(* Logix 5000 project; controller LeakTestAuto vendor 1 type 14 code 226 rev 37.11; software revision 37.01; part 6 of 12 *)
(* tags used below, declared in another part *)
   AOI_CTS1 : AOI_CTS_INSTRUMENT;
   AOI_CTS2 : AOI_CTS_INSTRUMENT;
   AOI_OP220_Seq : AOI_Sequencer_x64;
   AOI_RobotPos : AOI_RobotPositions;
   AOI_SeqSteps : AOI_StandardSeqSteps;
   AOI_SRX100 : AOI_KeyenceBarcode;
   Barcode_ResultData : STR_Barcode;
   BarcodeBypass : BOOL;
   BarcodeInputs : udt_KeyenceScannerInputs;
   BarcodeScanner : udt_OutputStructure;
   Conveyor : udt_OutputStructure;
   Conveyor_Seq : udt_SequenceStructure_X64;
   ConveyorHomeCounter : COUNTER;
   CurrentDUTData : udt_DUTHistory[2];
   DryCycle_N1Ready : BOOL;
   DryCycle_N2Ready : BOOL;
   DUTHistoryDump : udt_DUTHistory;
   DUTTestHistory : udt_DUTHistory[10];
   FFLU_DUTHistory : CONTROL;
   InfeedCounter : COUNTER;
   LeakTester1 : udt_OutputStructure;
   LeakTester2 : udt_OutputStructure;
   Nest1Bypass : BOOL;
   Nest1Cylinder : udt_OutputStructure;
   Nest1Empty : BOOL;
   Nest1Ready : BOOL;
   Nest2Bypass : BOOL;
   Nest2Cylinder : udt_OutputStructure;
   Nest2Empty : BOOL;
   Nest2Ready : BOOL;
   OP220 : udt_Mode;
   OP220_HomingSeq : udt_SequenceStructure_X64;
   OP220_Seq : udt_SequenceStructure_X64;
   OutfeedCounter : COUNTER;
   ResetFeedCounters : BOOL;
   RFID_TagStatus : BOOL[32];
   RFIDLoadingNestScanner : udt_OutputStructure;
   RFIDScanner : udt_OutputStructure;
   Robot : udt_OutputStructure;
   RobotGripper : udt_OutputStructure;
   RobotInputs : udt_EpsonInputs;
   TON_ConvUnloadDelay : TIMER;
   Delay_TMR : TIMER[11];   // Delay Timers
   I_OP220_N3_CONVEYOR_LOAD : ALIAS FOR Local:3:I.Pt12.Data;
   I_OP220_N3_CONVEYOR_UNLOAD : ALIAS FOR Local:3:I.Pt14.Data;
   I_OP220_N3_DUT_PRE_NEST_0 : ALIAS FOR Local:3:I.Pt00.Data;
   I_OP220_N3_DUT_PRE_NEST_1 : ALIAS FOR Local:3:I.Pt01.Data;
   I_OP220_N3_DUT_PRE_NEST_2 : ALIAS FOR Local:3:I.Pt02.Data;
   I_OP220_N3_NEST1_EXTEND : ALIAS FOR Local:3:I.Pt04.Data;
   I_OP220_N3_NEST1_HOME : ALIAS FOR Local:3:I.Pt03.Data;
   I_OP220_N3_NEST2_EXTEND : ALIAS FOR Local:3:I.Pt06.Data;
   I_OP220_N3_NEST2_HOME : ALIAS FOR Local:3:I.Pt05.Data;
   Ignition_Bypass : BOOL;
   James_Dint : DINT;   // James Test Word
   null : STRING;
   PLC : AOI_PLC;
   ST1_Ignition_DataReady : BOOL;
   ST1_Ignition_DataReady_Setup : BOOL;
   ST1_Ignition_DataReceived : BOOL;
   ST1_Ignition_SerialNum : STRING;
   ST1_Ignition_Status : DINT;
   ST2_Ignition_DataReady : BOOL;
   ST2_Ignition_DataReady_Setup : BOOL;
   ST2_Ignition_DataReceived : BOOL;
   ST2_Ignition_SerialNum : STRING;
   ST2_Ignition_Status : DINT;
(* MainProgram, continued *)

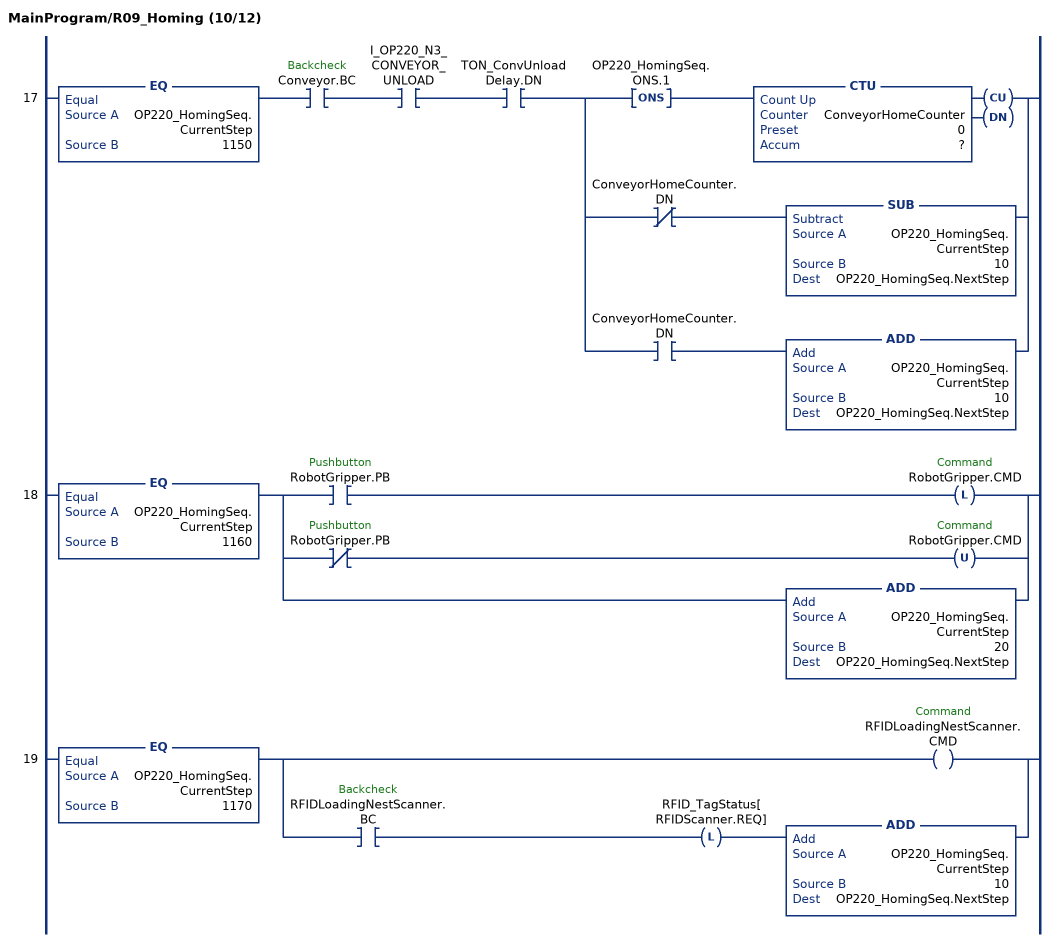
   [picture p62: MainProgram/R09_Homing rungs 17-19]
   17: EQ(OP220_HomingSeq.CurrentStep,1150)XIC(Conveyor.BC)XIC(I_OP220_N3_CONVEYOR_UNLOAD)XIC(TON_ConvUnloadDelay.DN)[ONS(OP220_HomingSeq.ONS.1) CTU(ConveyorHomeCounter,?,?) ,[XIO(ConveyorHomeCounter.DN) SUB(OP220_HomingSeq.CurrentStep,10,OP220_HomingSeq.NextStep) ,XIC(ConveyorHomeCounter.DN) ADD(OP220_HomingSeq.CurrentStep,10,OP220_HomingSeq.NextStep) ] ];
   18: EQ(OP220_HomingSeq.CurrentStep,1160)[XIC(RobotGripper.PB) OTL(RobotGripper.CMD) ,XIO(RobotGripper.PB) OTU(RobotGripper.CMD) ,ADD(OP220_HomingSeq.CurrentStep,20,OP220_HomingSeq.NextStep) ];
   19: EQ(OP220_HomingSeq.CurrentStep,1170)[OTE(RFIDLoadingNestScanner.CMD) ,XIC(RFIDLoadingNestScanner.BC) OTL(RFID_TagStatus[RFIDScanner.REQ]) ADD(OP220_HomingSeq.CurrentStep,10,OP220_HomingSeq.NextStep) ];
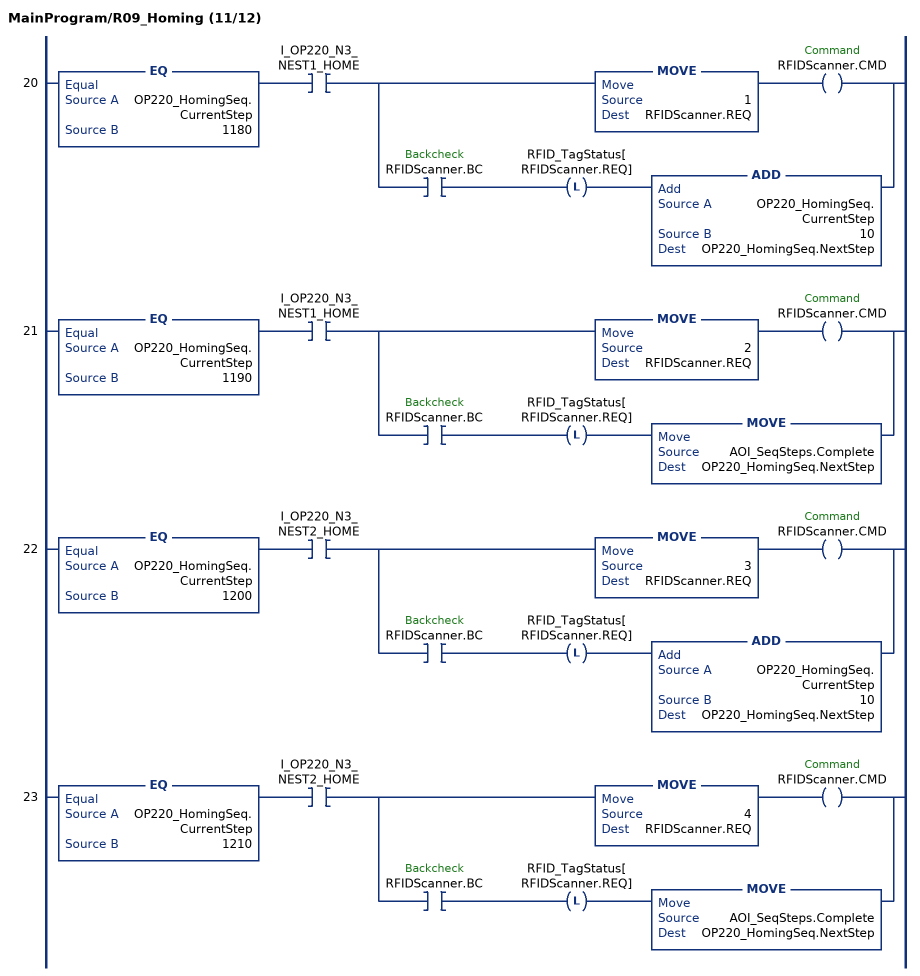
   20: EQ(OP220_HomingSeq.CurrentStep,1180)XIC(I_OP220_N3_NEST1_HOME)[MOVE(1,RFIDScanner.REQ) OTE(RFIDScanner.CMD) ,XIC(RFIDScanner.BC) OTL(RFID_TagStatus[RFIDScanner.REQ]) ADD(OP220_HomingSeq.CurrentStep,10,OP220_HomingSeq.NextStep) ];
   21: EQ(OP220_HomingSeq.CurrentStep,1190)XIC(I_OP220_N3_NEST1_HOME)[MOVE(2,RFIDScanner.REQ) OTE(RFIDScanner.CMD) ,XIC(RFIDScanner.BC) OTL(RFID_TagStatus[RFIDScanner.REQ]) MOVE(AOI_SeqSteps.Complete,OP220_HomingSeq.NextStep) ];
   22: EQ(OP220_HomingSeq.CurrentStep,1200)XIC(I_OP220_N3_NEST2_HOME)[MOVE(3,RFIDScanner.REQ) OTE(RFIDScanner.CMD) ,XIC(RFIDScanner.BC) OTL(RFID_TagStatus[RFIDScanner.REQ]) ADD(OP220_HomingSeq.CurrentStep,10,OP220_HomingSeq.NextStep) ];
   23: EQ(OP220_HomingSeq.CurrentStep,1210)XIC(I_OP220_N3_NEST2_HOME)[MOVE(4,RFIDScanner.REQ) OTE(RFIDScanner.CMD) ,XIC(RFIDScanner.BC) OTL(RFID_TagStatus[RFIDScanner.REQ]) MOVE(AOI_SeqSteps.Complete,OP220_HomingSeq.NextStep) ];
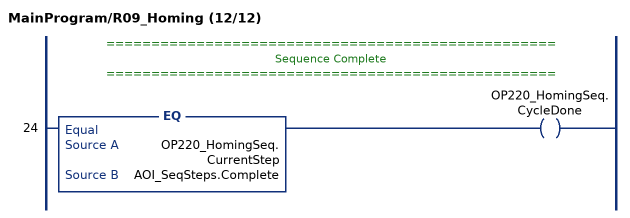
   // ==================================================
   // Sequence Complete
   // ==================================================
   24: EQ(OP220_HomingSeq.CurrentStep,AOI_SeqSteps.Complete)OTE(OP220_HomingSeq.CycleDone);
END_ROUTINE

ROUTINE R10_Sequence   (* ladder *)
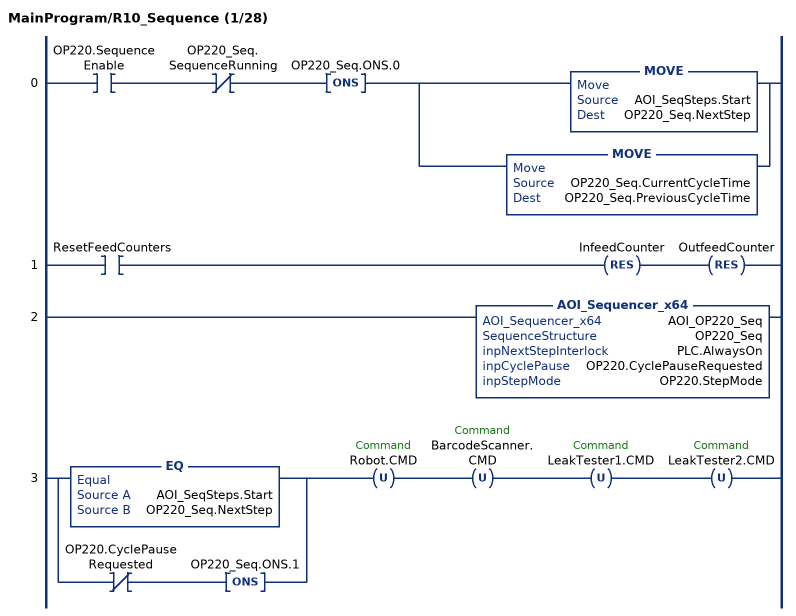
   0: XIC(OP220.SequenceEnable)XIO(OP220_Seq.SequenceRunning)ONS(OP220_Seq.ONS.0)[MOVE(AOI_SeqSteps.Start,OP220_Seq.NextStep) ,MOVE(OP220_Seq.CurrentCycleTime,OP220_Seq.PreviousCycleTime) ];
   1: XIC(ResetFeedCounters)RES(InfeedCounter)RES(OutfeedCounter);
   2: AOI_Sequencer_x64(AOI_OP220_Seq,OP220_Seq,PLC.AlwaysOn,OP220.CyclePauseRequested,OP220.StepMode);
   3: [EQ(AOI_SeqSteps.Start,OP220_Seq.NextStep) ,XIO(OP220.CyclePauseRequested) ONS(OP220_Seq.ONS.1) ]OTU(Robot.CMD)OTU(BarcodeScanner.CMD)OTU(LeakTester1.CMD)OTU(LeakTester2.CMD);
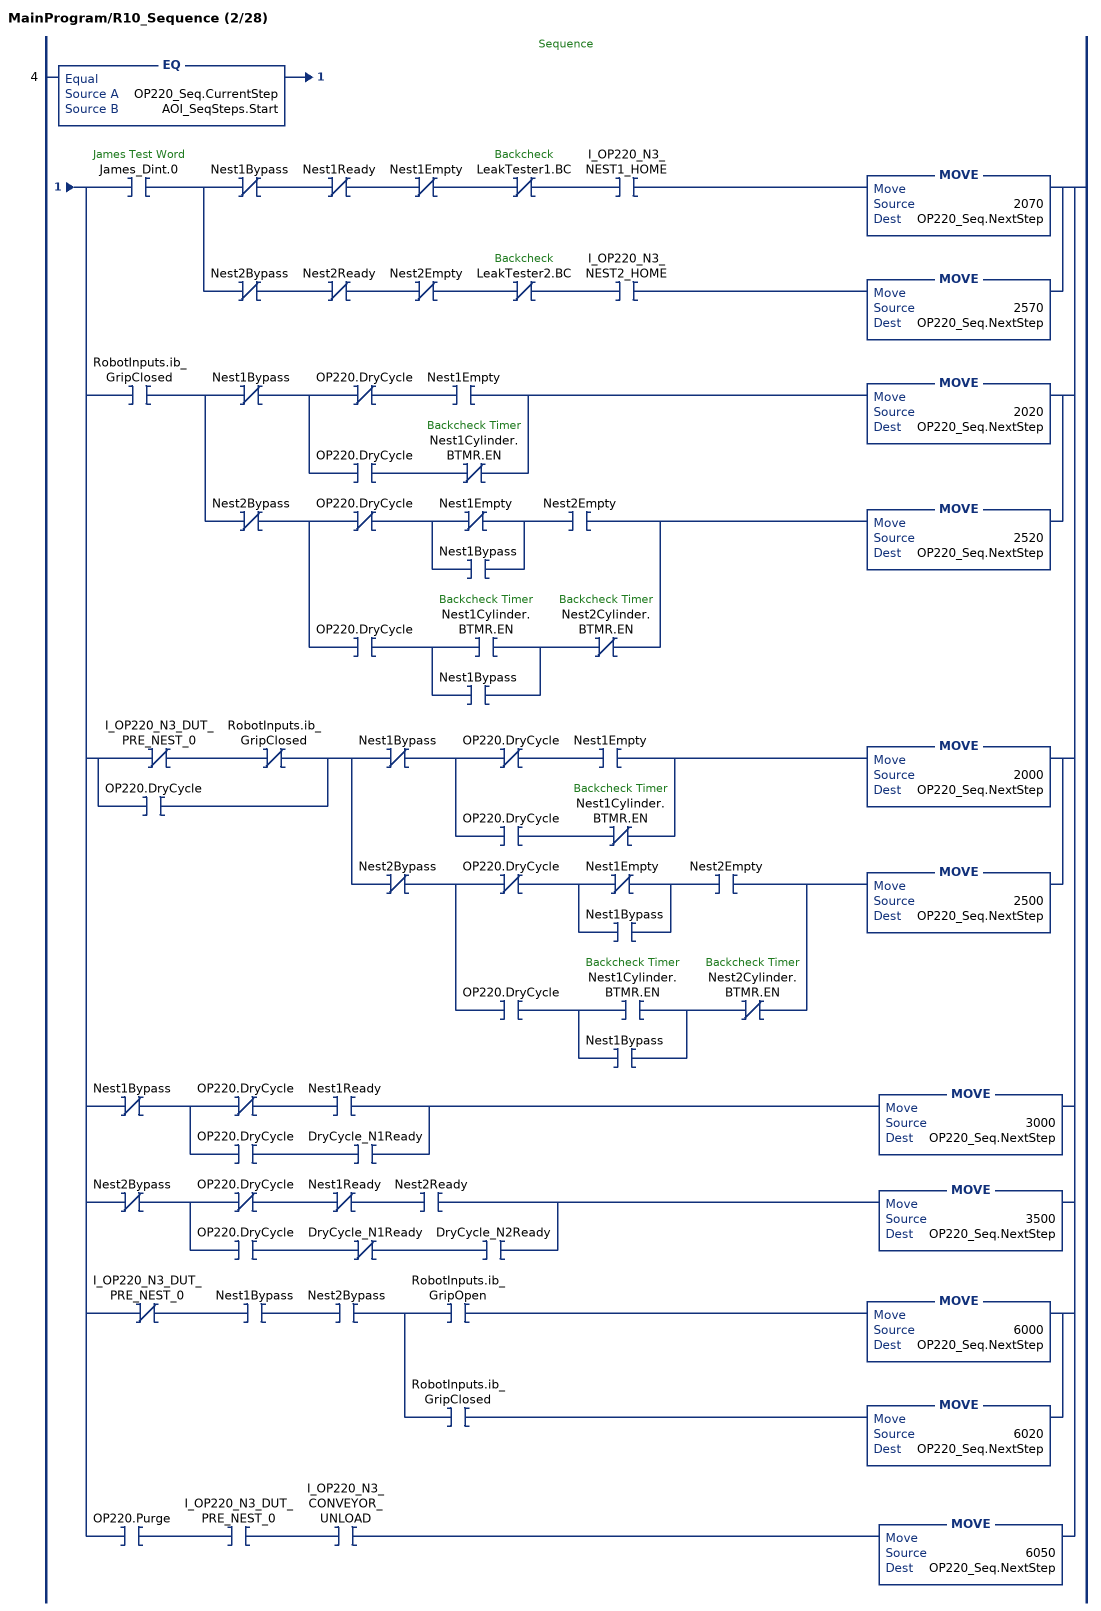
   // Sequence
   4: EQ(OP220_Seq.CurrentStep,AOI_SeqSteps.Start)[XIC(James_Dint.0) [XIO(Nest1Bypass) XIO(Nest1Ready) XIO(Nest1Empty) XIO(LeakTester1.BC) XIC(I_OP220_N3_NEST1_HOME) MOVE(2070,OP220_Seq.NextStep) ,XIO(Nest2Bypass) XIO(Nest2Ready) XIO(Nest2Empty) XIO(LeakTester2.BC) XIC(I_OP220_N3_NEST2_HOME) MOVE(2570,OP220_Seq.NextStep) ] ,XIC(RobotInputs.ib_GripClosed) [XIO(Nest1Bypass) [XIO(OP220.DryCycle) XIC(Nest1Empty) ,XIC(OP220.DryCycle) XIO(Nest1Cylinder.BTMR.EN) ] MOVE(2020,OP220_Seq.NextStep) ,XIO(Nest2Bypass) [XIO(OP220.DryCycle) [XIO(Nest1Empty) ,XIC(Nest1Bypass) ] XIC(Nest2Empty) ,XIC(OP220.DryCycle) [XIC(Nest1Cylinder.BTMR.EN) ,XIC(Nest1Bypass) ] XIO(Nest2Cylinder.BTMR.EN) ] MOVE(2520,OP220_Seq.NextStep) ] ,[XIO(I_OP220_N3_DUT_PRE_NEST_0) XIO(RobotInputs.ib_GripClosed) ,XIC(OP220.DryCycle) ] [XIO(Nest1Bypass) [XIO(OP220.DryCycle) XIC(Nest1Empty) ,XIC(OP220.DryCycle) XIO(Nest1Cylinder.BTMR.EN) ] MOVE(2000,OP220_Seq.NextStep) ,XIO(Nest2Bypass) [XIO(OP220.DryCycle) [XIO(Nest1Empty) ,XIC(Nest1Bypass) ] XIC(Nest2Empty) ,XIC(OP220.DryCycle) [XIC(Nest1Cylinder.BTMR.EN) ,XIC(Nest1Bypass) ] XIO(Nest2Cylinder.BTMR.EN) ] MOVE(2500,OP220_Seq.NextStep) ] ,[XIO(Nest1Bypass) [XIO(OP220.DryCycle) XIC(Nest1Ready) ,XIC(OP220.DryCycle) XIC(DryCycle_N1Ready) ] MOVE(3000,OP220_Seq.NextStep) ,XIO(Nest2Bypass) [XIO(OP220.DryCycle) XIO(Nest1Ready) XIC(Nest2Ready) ,XIC(OP220.DryCycle) XIO(DryCycle_N1Ready) XIC(DryCycle_N2Ready) ] MOVE(3500,OP220_Seq.NextStep) ] ,XIO(I_OP220_N3_DUT_PRE_NEST_0) XIC(Nest1Bypass) XIC(Nest2Bypass) [XIC(RobotInputs.ib_GripOpen) MOVE(6000,OP220_Seq.NextStep) ,XIC(RobotInputs.ib_GripClosed) MOVE(6020,OP220_Seq.NextStep) ] ,XIC(OP220.Purge) XIC(I_OP220_N3_DUT_PRE_NEST_0) XIC(I_OP220_N3_CONVEYOR_UNLOAD) MOVE(6050,OP220_Seq.NextStep) ];
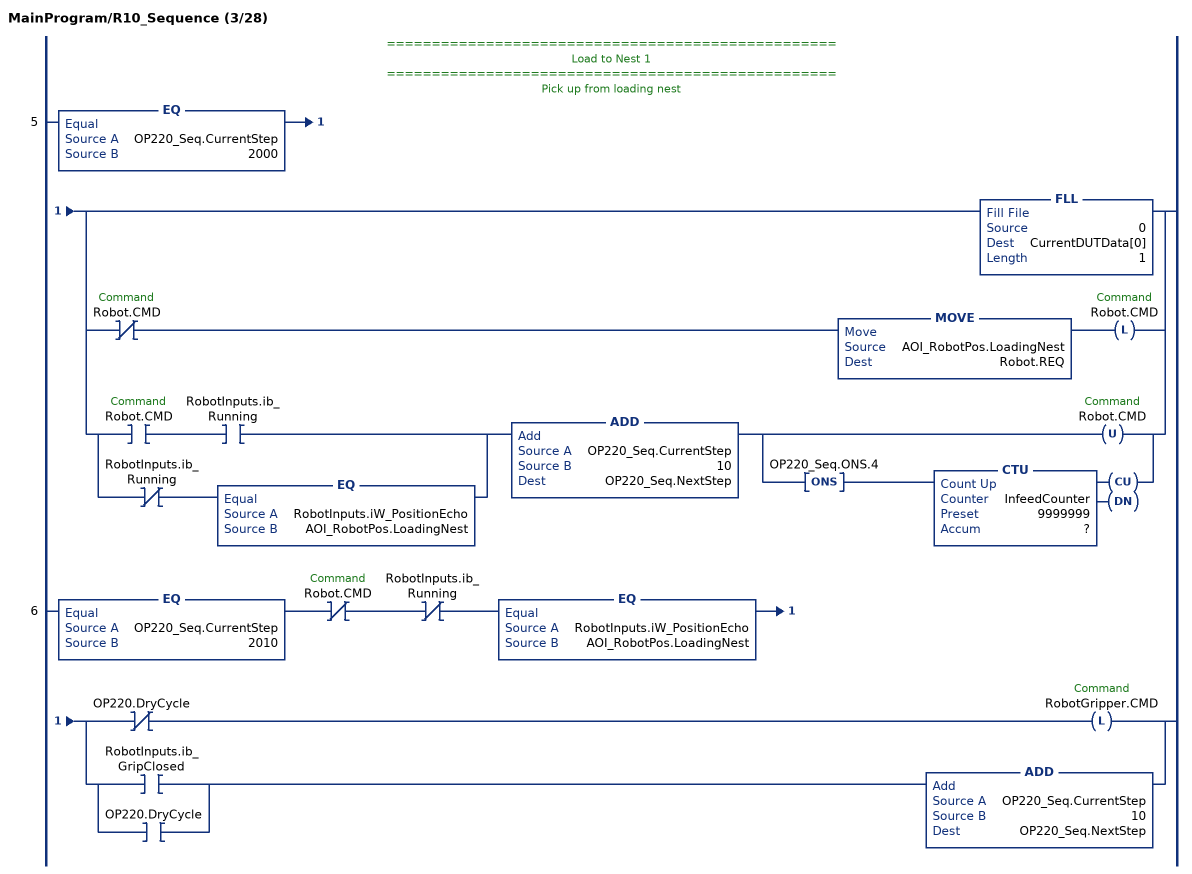
   // ==================================================
   // Load to Nest 1
   // ==================================================
   // Pick up from loading nest
   5: EQ(OP220_Seq.CurrentStep,2000)[FLL(0,CurrentDUTData[0],1) ,XIO(Robot.CMD) MOVE(AOI_RobotPos.LoadingNest,Robot.REQ) OTL(Robot.CMD) ,[XIC(Robot.CMD) XIC(RobotInputs.ib_Running) ,XIO(RobotInputs.ib_Running) EQ(RobotInputs.iW_PositionEcho,AOI_RobotPos.LoadingNest) ] ADD(OP220_Seq.CurrentStep,10,OP220_Seq.NextStep) [OTU(Robot.CMD) ,ONS(OP220_Seq.ONS.4) CTU(InfeedCounter,?,?) ] ];
   6: EQ(OP220_Seq.CurrentStep,2010)XIO(Robot.CMD)XIO(RobotInputs.ib_Running)EQ(RobotInputs.iW_PositionEcho,AOI_RobotPos.LoadingNest)[XIO(OP220.DryCycle) OTL(RobotGripper.CMD) ,[XIC(RobotInputs.ib_GripClosed) ,XIC(OP220.DryCycle) ] ADD(OP220_Seq.CurrentStep,10,OP220_Seq.NextStep) ];
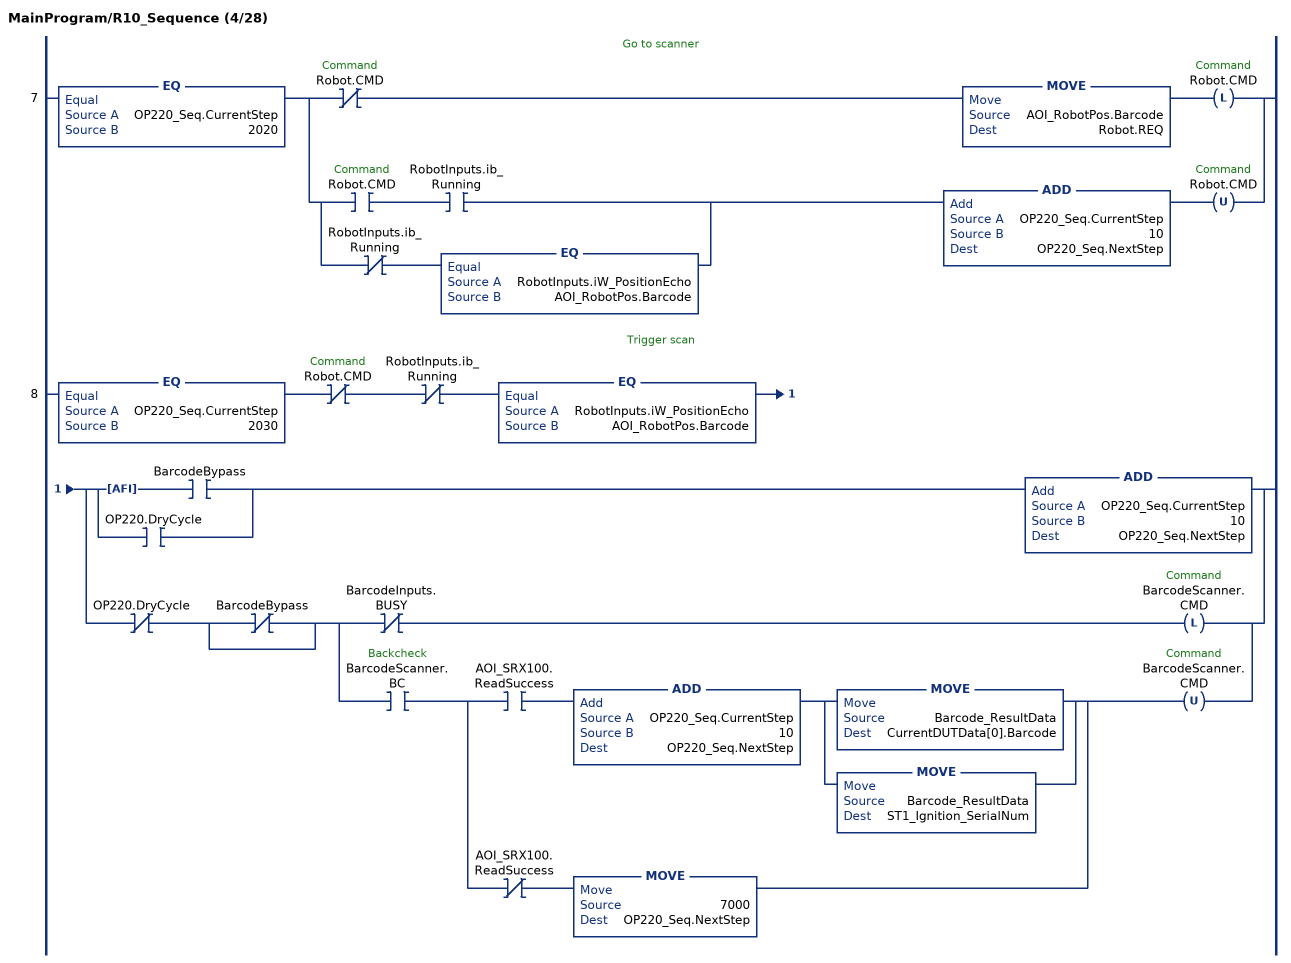
   // Go to scanner
   7: EQ(OP220_Seq.CurrentStep,2020)[XIO(Robot.CMD) MOVE(AOI_RobotPos.Barcode,Robot.REQ) OTL(Robot.CMD) ,[XIC(Robot.CMD) XIC(RobotInputs.ib_Running) ,XIO(RobotInputs.ib_Running) EQ(RobotInputs.iW_PositionEcho,AOI_RobotPos.Barcode) ] ADD(OP220_Seq.CurrentStep,10,OP220_Seq.NextStep) OTU(Robot.CMD) ];
   // Trigger scan
   8: EQ(OP220_Seq.CurrentStep,2030)XIO(Robot.CMD)XIO(RobotInputs.ib_Running)EQ(RobotInputs.iW_PositionEcho,AOI_RobotPos.Barcode)[[AFI() XIC(BarcodeBypass) ,XIC(OP220.DryCycle) ] ADD(OP220_Seq.CurrentStep,10,OP220_Seq.NextStep) ,XIO(OP220.DryCycle) [XIO(BarcodeBypass) ,] [XIO(BarcodeInputs.BUSY) OTL(BarcodeScanner.CMD) ,XIC(BarcodeScanner.BC) [XIC(AOI_SRX100.ReadSuccess) ADD(OP220_Seq.CurrentStep,10,OP220_Seq.NextStep) [MOVE(Barcode_ResultData,CurrentDUTData[0].Barcode) ,MOVE(Barcode_ResultData,ST1_Ignition_SerialNum) ] ,XIO(AOI_SRX100.ReadSuccess) MOVE(7000,OP220_Seq.NextStep) ] OTU(BarcodeScanner.CMD) ] ];
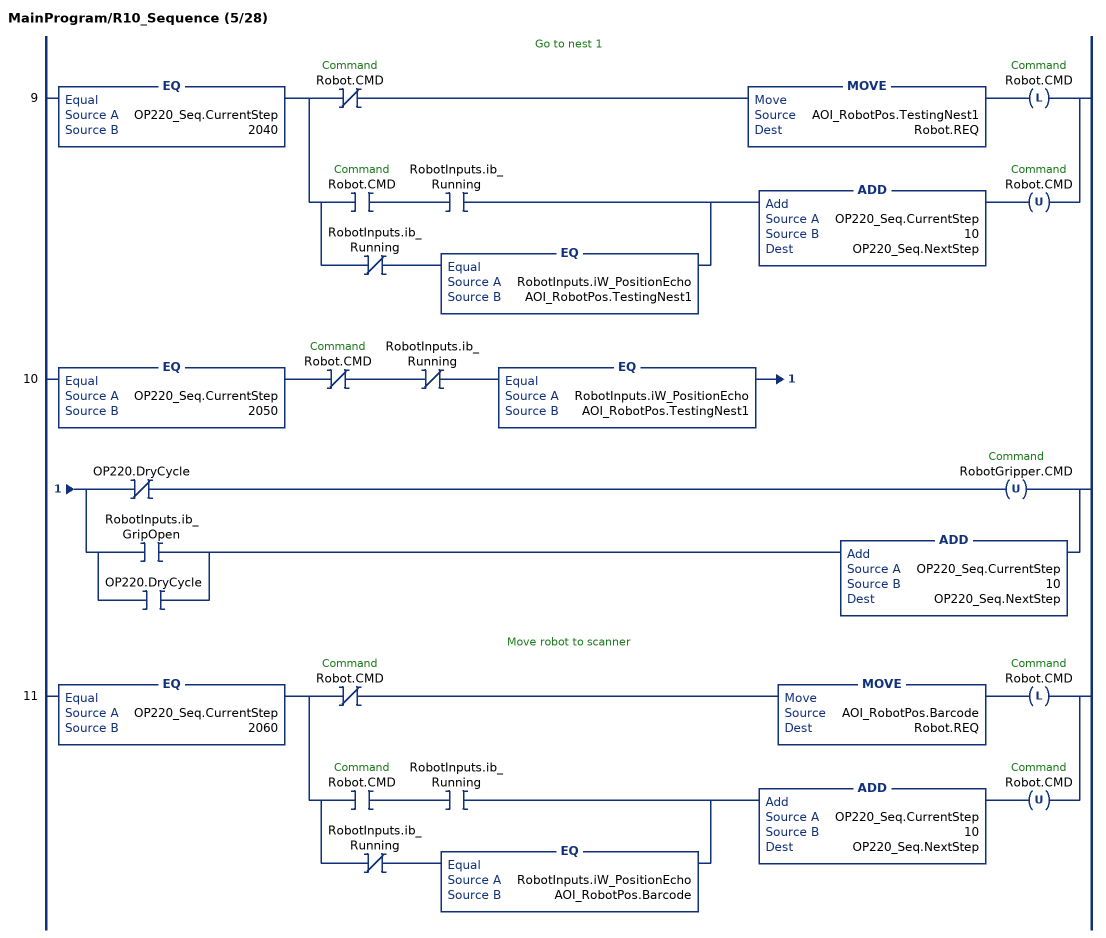
   // Go to nest 1
   9: EQ(OP220_Seq.CurrentStep,2040)[XIO(Robot.CMD) MOVE(AOI_RobotPos.TestingNest1,Robot.REQ) OTL(Robot.CMD) ,[XIC(Robot.CMD) XIC(RobotInputs.ib_Running) ,XIO(RobotInputs.ib_Running) EQ(RobotInputs.iW_PositionEcho,AOI_RobotPos.TestingNest1) ] ADD(OP220_Seq.CurrentStep,10,OP220_Seq.NextStep) OTU(Robot.CMD) ];
   10: EQ(OP220_Seq.CurrentStep,2050)XIO(Robot.CMD)XIO(RobotInputs.ib_Running)EQ(RobotInputs.iW_PositionEcho,AOI_RobotPos.TestingNest1)[XIO(OP220.DryCycle) OTU(RobotGripper.CMD) ,[XIC(RobotInputs.ib_GripOpen) ,XIC(OP220.DryCycle) ] ADD(OP220_Seq.CurrentStep,10,OP220_Seq.NextStep) ];
   // Move robot to scanner
   11: EQ(OP220_Seq.CurrentStep,2060)[XIO(Robot.CMD) MOVE(AOI_RobotPos.Barcode,Robot.REQ) OTL(Robot.CMD) ,[XIC(Robot.CMD) XIC(RobotInputs.ib_Running) ,XIO(RobotInputs.ib_Running) EQ(RobotInputs.iW_PositionEcho,AOI_RobotPos.Barcode) ] ADD(OP220_Seq.CurrentStep,10,OP220_Seq.NextStep) OTU(Robot.CMD) ];
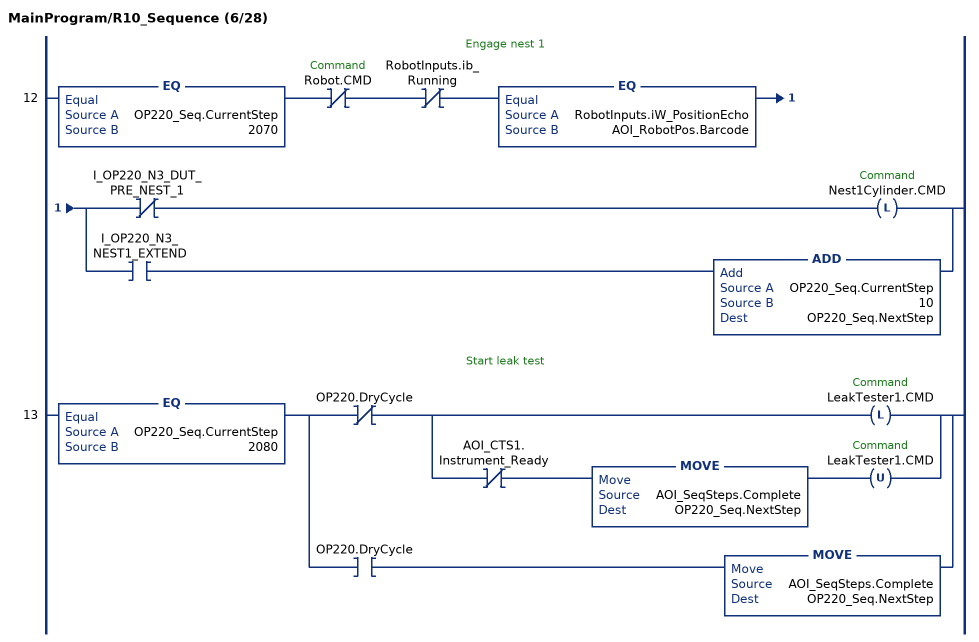
   // Engage nest 1
   12: EQ(OP220_Seq.CurrentStep,2070)XIO(Robot.CMD)XIO(RobotInputs.ib_Running)EQ(RobotInputs.iW_PositionEcho,AOI_RobotPos.Barcode)[XIO(I_OP220_N3_DUT_PRE_NEST_1) OTL(Nest1Cylinder.CMD) ,XIC(I_OP220_N3_NEST1_EXTEND) ADD(OP220_Seq.CurrentStep,10,OP220_Seq.NextStep) ];
   // Start leak test
   13: EQ(OP220_Seq.CurrentStep,2080)[XIO(OP220.DryCycle) [OTL(LeakTester1.CMD) ,XIO(AOI_CTS1.Instrument_Ready) MOVE(AOI_SeqSteps.Complete,OP220_Seq.NextStep) OTU(LeakTester1.CMD) ] ,XIC(OP220.DryCycle) MOVE(AOI_SeqSteps.Complete,OP220_Seq.NextStep) ];
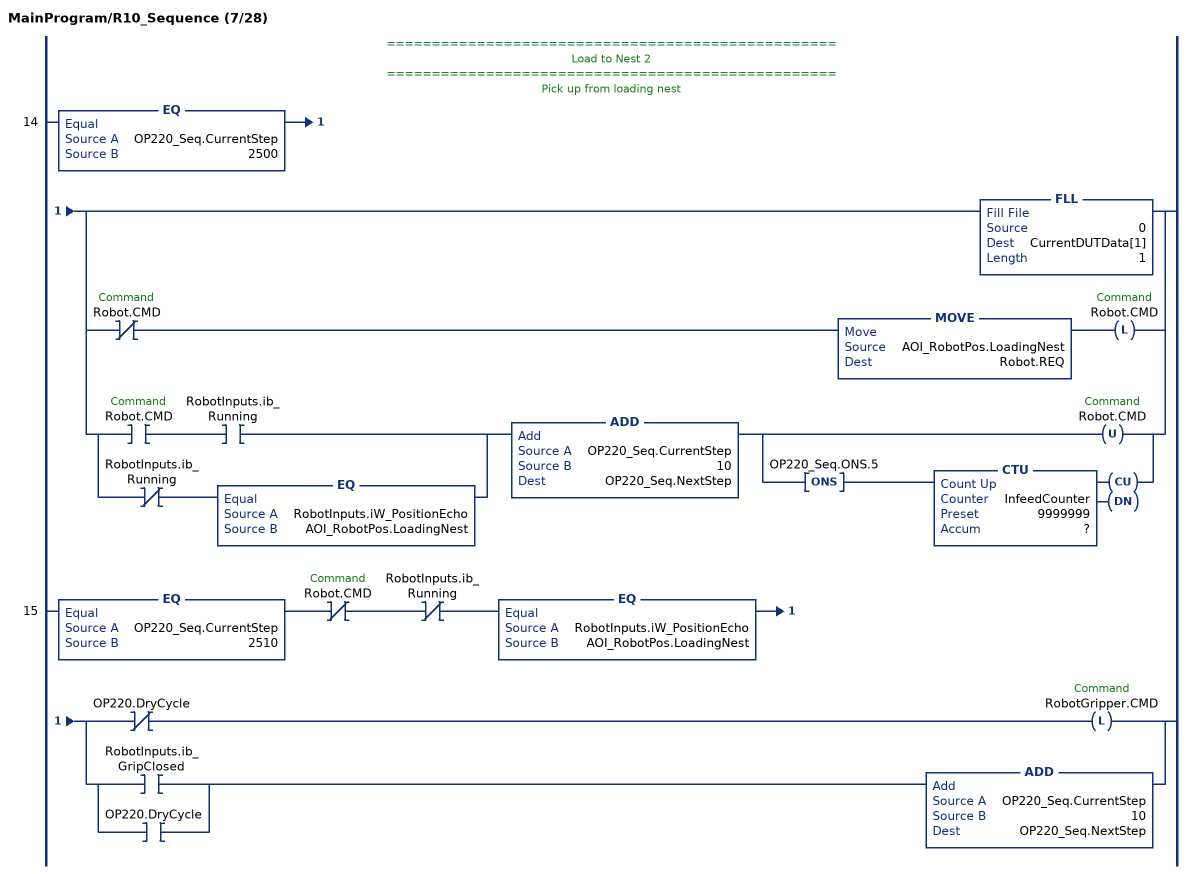
   // ==================================================
   // Load to Nest 2
   // ==================================================
   // Pick up from loading nest
   14: EQ(OP220_Seq.CurrentStep,2500)[FLL(0,CurrentDUTData[1],1) ,XIO(Robot.CMD) MOVE(AOI_RobotPos.LoadingNest,Robot.REQ) OTL(Robot.CMD) ,[XIC(Robot.CMD) XIC(RobotInputs.ib_Running) ,XIO(RobotInputs.ib_Running) EQ(RobotInputs.iW_PositionEcho,AOI_RobotPos.LoadingNest) ] ADD(OP220_Seq.CurrentStep,10,OP220_Seq.NextStep) [OTU(Robot.CMD) ,ONS(OP220_Seq.ONS.5) CTU(InfeedCounter,?,?) ] ];
   15: EQ(OP220_Seq.CurrentStep,2510)XIO(Robot.CMD)XIO(RobotInputs.ib_Running)EQ(RobotInputs.iW_PositionEcho,AOI_RobotPos.LoadingNest)[XIO(OP220.DryCycle) OTL(RobotGripper.CMD) ,[XIC(RobotInputs.ib_GripClosed) ,XIC(OP220.DryCycle) ] ADD(OP220_Seq.CurrentStep,10,OP220_Seq.NextStep) ];
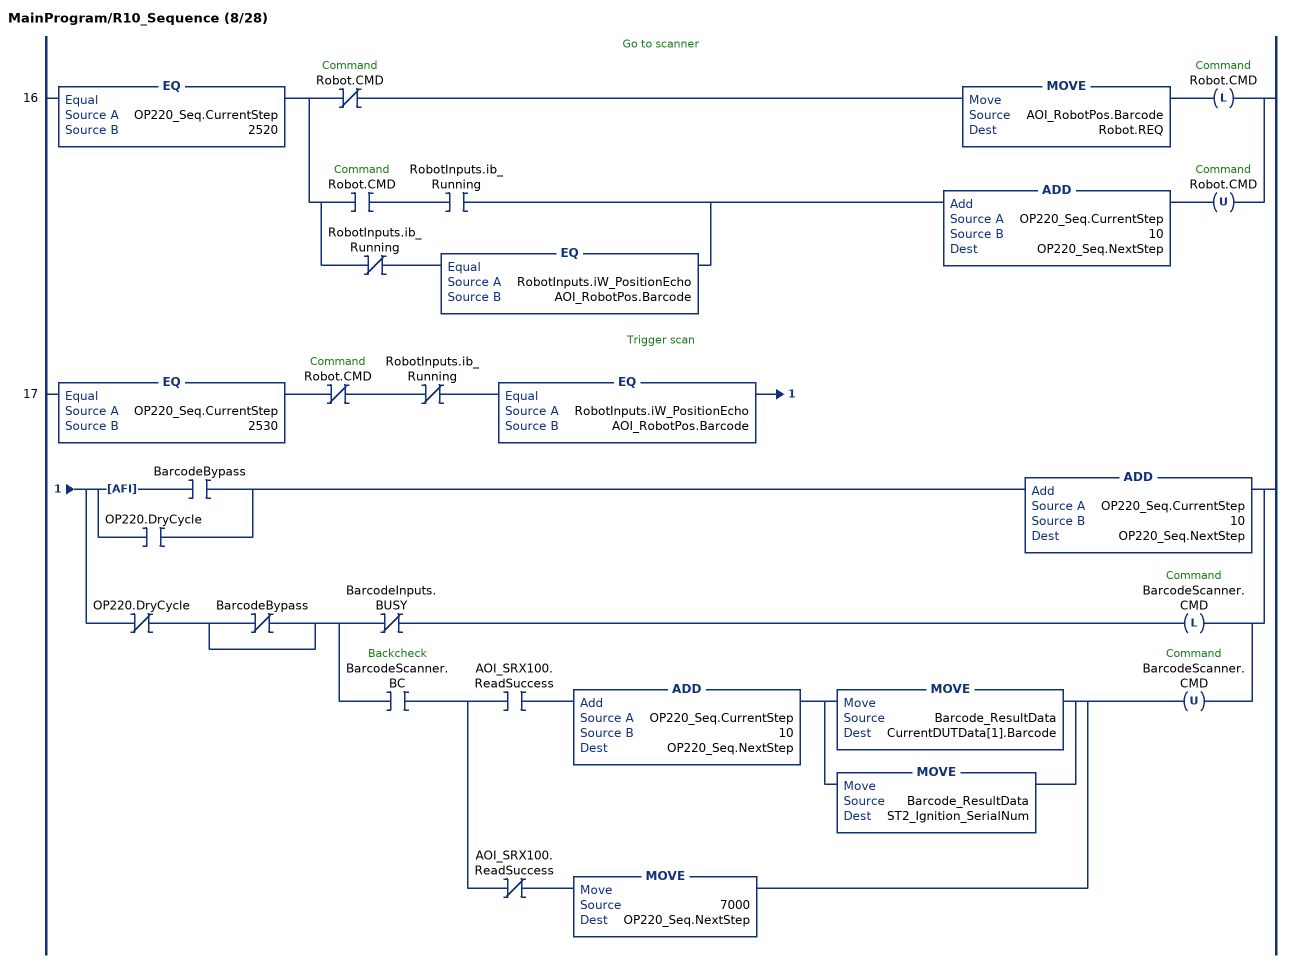
   // Go to scanner
   16: EQ(OP220_Seq.CurrentStep,2520)[XIO(Robot.CMD) MOVE(AOI_RobotPos.Barcode,Robot.REQ) OTL(Robot.CMD) ,[XIC(Robot.CMD) XIC(RobotInputs.ib_Running) ,XIO(RobotInputs.ib_Running) EQ(RobotInputs.iW_PositionEcho,AOI_RobotPos.Barcode) ] ADD(OP220_Seq.CurrentStep,10,OP220_Seq.NextStep) OTU(Robot.CMD) ];
   // Trigger scan
   17: EQ(OP220_Seq.CurrentStep,2530)XIO(Robot.CMD)XIO(RobotInputs.ib_Running)EQ(RobotInputs.iW_PositionEcho,AOI_RobotPos.Barcode)[[AFI() XIC(BarcodeBypass) ,XIC(OP220.DryCycle) ] ADD(OP220_Seq.CurrentStep,10,OP220_Seq.NextStep) ,XIO(OP220.DryCycle) [XIO(BarcodeBypass) ,] [XIO(BarcodeInputs.BUSY) OTL(BarcodeScanner.CMD) ,XIC(BarcodeScanner.BC) [XIC(AOI_SRX100.ReadSuccess) ADD(OP220_Seq.CurrentStep,10,OP220_Seq.NextStep) [MOVE(Barcode_ResultData,CurrentDUTData[1].Barcode) ,MOVE(Barcode_ResultData,ST2_Ignition_SerialNum) ] ,XIO(AOI_SRX100.ReadSuccess) MOVE(7000,OP220_Seq.NextStep) ] OTU(BarcodeScanner.CMD) ] ];
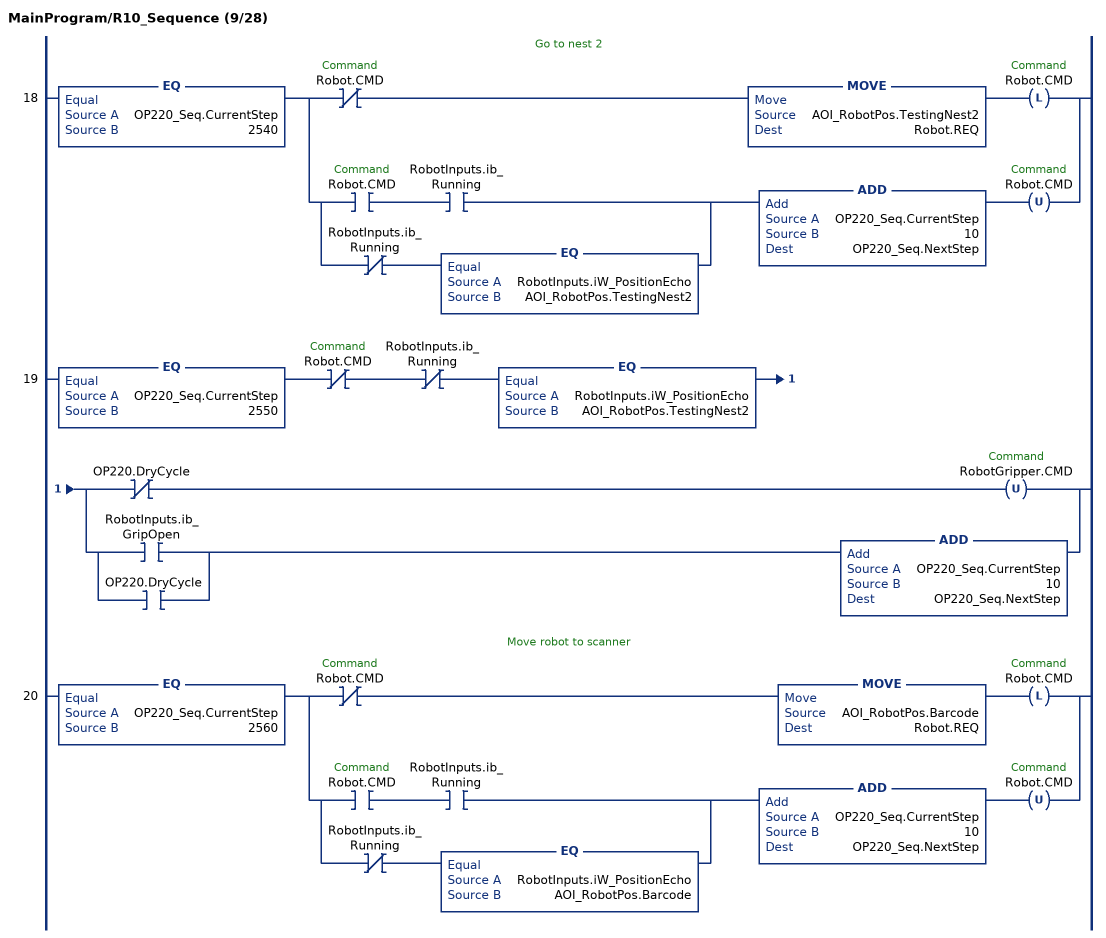
   // Go to nest 2
   18: EQ(OP220_Seq.CurrentStep,2540)[XIO(Robot.CMD) MOVE(AOI_RobotPos.TestingNest2,Robot.REQ) OTL(Robot.CMD) ,[XIC(Robot.CMD) XIC(RobotInputs.ib_Running) ,XIO(RobotInputs.ib_Running) EQ(RobotInputs.iW_PositionEcho,AOI_RobotPos.TestingNest2) ] ADD(OP220_Seq.CurrentStep,10,OP220_Seq.NextStep) OTU(Robot.CMD) ];
   19: EQ(OP220_Seq.CurrentStep,2550)XIO(Robot.CMD)XIO(RobotInputs.ib_Running)EQ(RobotInputs.iW_PositionEcho,AOI_RobotPos.TestingNest2)[XIO(OP220.DryCycle) OTU(RobotGripper.CMD) ,[XIC(RobotInputs.ib_GripOpen) ,XIC(OP220.DryCycle) ] ADD(OP220_Seq.CurrentStep,10,OP220_Seq.NextStep) ];
   // Move robot to scanner
   20: EQ(OP220_Seq.CurrentStep,2560)[XIO(Robot.CMD) MOVE(AOI_RobotPos.Barcode,Robot.REQ) OTL(Robot.CMD) ,[XIC(Robot.CMD) XIC(RobotInputs.ib_Running) ,XIO(RobotInputs.ib_Running) EQ(RobotInputs.iW_PositionEcho,AOI_RobotPos.Barcode) ] ADD(OP220_Seq.CurrentStep,10,OP220_Seq.NextStep) OTU(Robot.CMD) ];
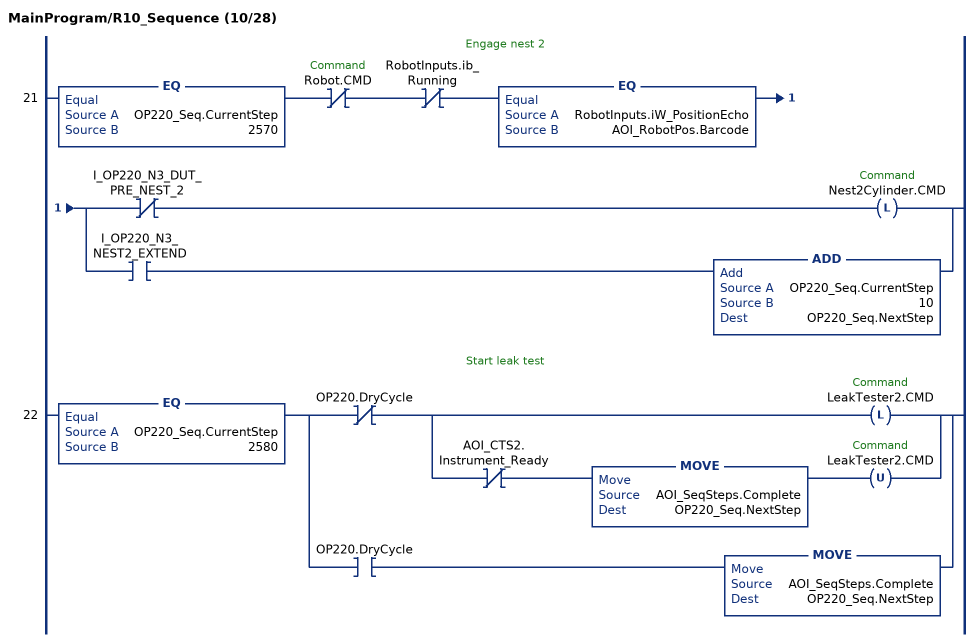
   // Engage nest 2
   21: EQ(OP220_Seq.CurrentStep,2570)XIO(Robot.CMD)XIO(RobotInputs.ib_Running)EQ(RobotInputs.iW_PositionEcho,AOI_RobotPos.Barcode)[XIO(I_OP220_N3_DUT_PRE_NEST_2) OTL(Nest2Cylinder.CMD) ,XIC(I_OP220_N3_NEST2_EXTEND) ADD(OP220_Seq.CurrentStep,10,OP220_Seq.NextStep) ];
   // Start leak test
   22: EQ(OP220_Seq.CurrentStep,2580)[XIO(OP220.DryCycle) [OTL(LeakTester2.CMD) ,XIO(AOI_CTS2.Instrument_Ready) MOVE(AOI_SeqSteps.Complete,OP220_Seq.NextStep) OTU(LeakTester2.CMD) ] ,XIC(OP220.DryCycle) MOVE(AOI_SeqSteps.Complete,OP220_Seq.NextStep) ];
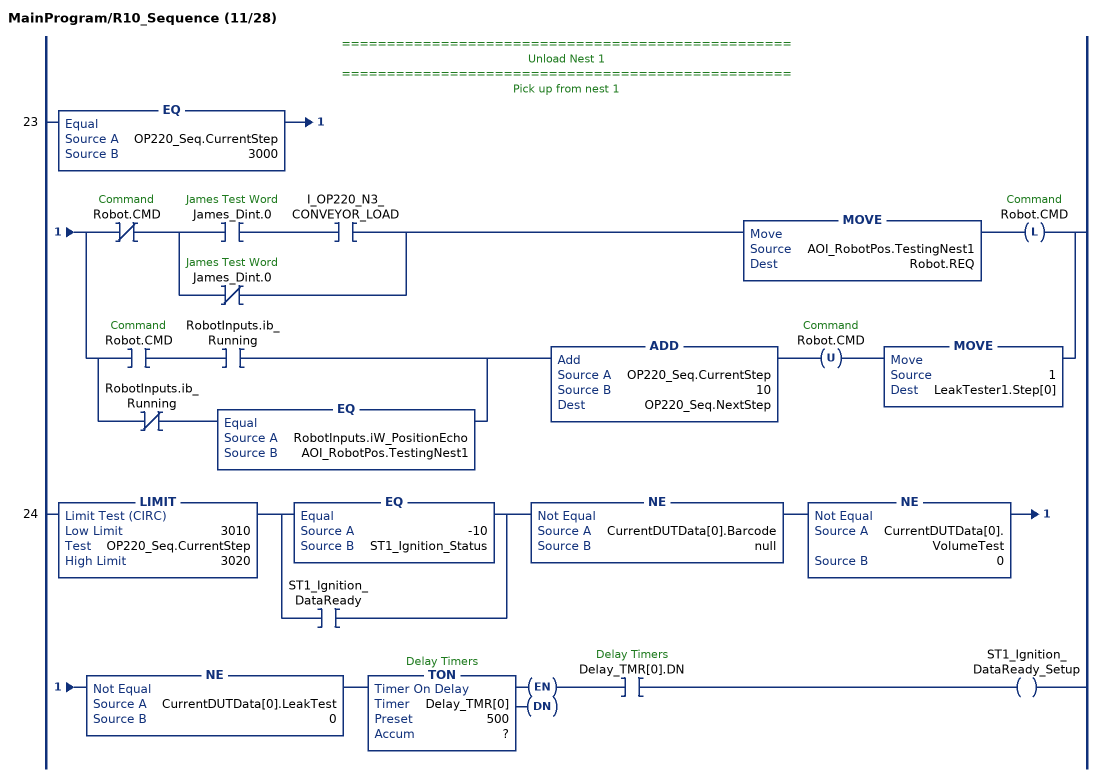
   // ==================================================
   // Unload Nest 1
   // ==================================================
   // Pick up from nest 1
   23: EQ(OP220_Seq.CurrentStep,3000)[XIO(Robot.CMD) [XIC(James_Dint.0) XIC(I_OP220_N3_CONVEYOR_LOAD) ,XIO(James_Dint.0) ] MOVE(AOI_RobotPos.TestingNest1,Robot.REQ) OTL(Robot.CMD) ,[XIC(Robot.CMD) XIC(RobotInputs.ib_Running) ,XIO(RobotInputs.ib_Running) EQ(RobotInputs.iW_PositionEcho,AOI_RobotPos.TestingNest1) ] ADD(OP220_Seq.CurrentStep,10,OP220_Seq.NextStep) OTU(Robot.CMD) MOVE(1,LeakTester1.Step[0]) ];
   24: LIMIT(3010,OP220_Seq.CurrentStep,3020)[EQ(-10,ST1_Ignition_Status) ,XIC(ST1_Ignition_DataReady) ]NE(CurrentDUTData[0].Barcode,null)NE(CurrentDUTData[0].VolumeTest,0)NE(CurrentDUTData[0].LeakTest,0)TON(Delay_TMR[0],?,?)XIC(Delay_TMR[0].DN)OTE(ST1_Ignition_DataReady_Setup);
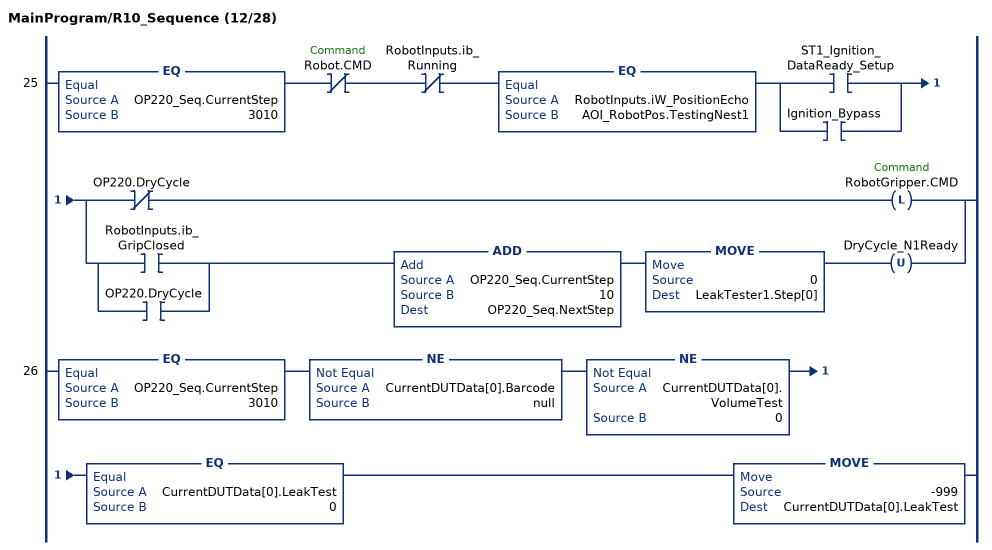
   25: EQ(OP220_Seq.CurrentStep,3010)XIO(Robot.CMD)XIO(RobotInputs.ib_Running)EQ(RobotInputs.iW_PositionEcho,AOI_RobotPos.TestingNest1)[XIC(ST1_Ignition_DataReady_Setup) ,XIC(Ignition_Bypass) ][XIO(OP220.DryCycle) OTL(RobotGripper.CMD) ,[XIC(RobotInputs.ib_GripClosed) ,XIC(OP220.DryCycle) ] ADD(OP220_Seq.CurrentStep,10,OP220_Seq.NextStep) MOVE(0,LeakTester1.Step[0]) OTU(DryCycle_N1Ready) ];
   26: EQ(OP220_Seq.CurrentStep,3010)NE(CurrentDUTData[0].Barcode,null)NE(CurrentDUTData[0].VolumeTest,0)EQ(CurrentDUTData[0].LeakTest,0)MOVE(-999,CurrentDUTData[0].LeakTest);
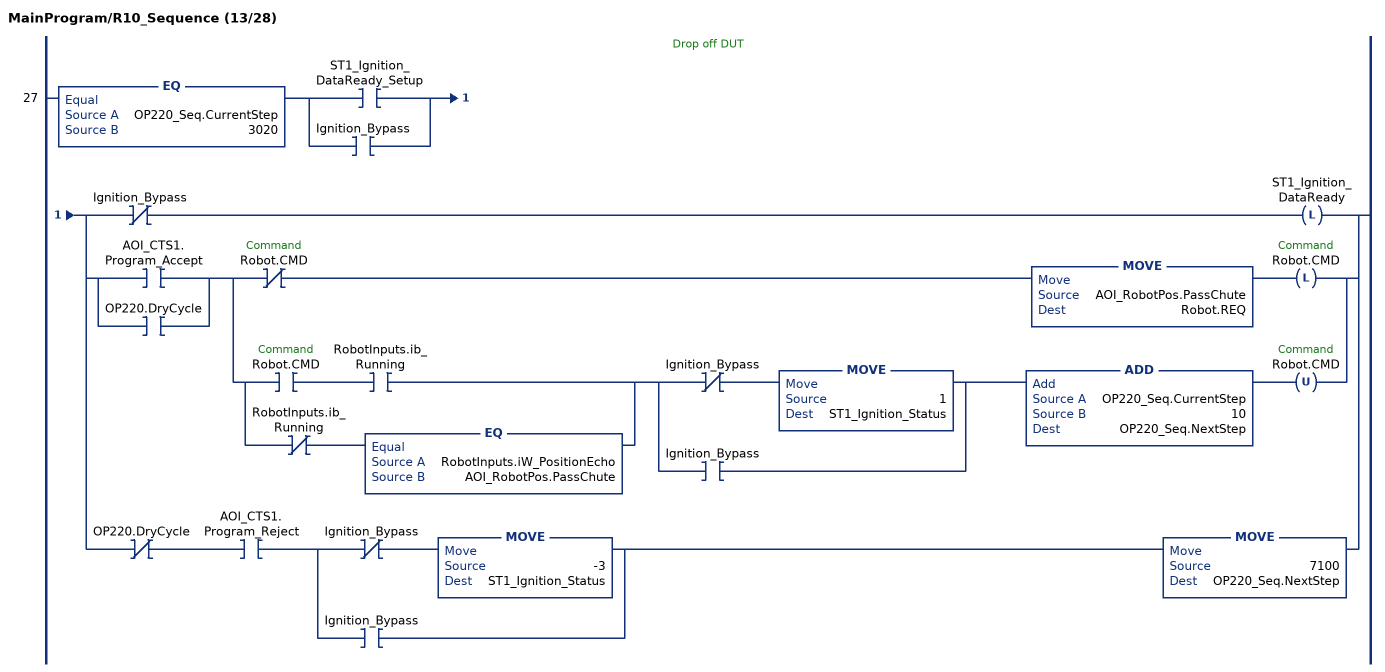
   // Drop off DUT
   27: EQ(OP220_Seq.CurrentStep,3020)[XIC(ST1_Ignition_DataReady_Setup) ,XIC(Ignition_Bypass) ][XIO(Ignition_Bypass) OTL(ST1_Ignition_DataReady) ,[XIC(AOI_CTS1.Program_Accept) ,XIC(OP220.DryCycle) ] [XIO(Robot.CMD) MOVE(AOI_RobotPos.PassChute,Robot.REQ) OTL(Robot.CMD) ,[XIC(Robot.CMD) XIC(RobotInputs.ib_Running) ,XIO(RobotInputs.ib_Running) EQ(RobotInputs.iW_PositionEcho,AOI_RobotPos.PassChute) ] [XIO(Ignition_Bypass) MOVE(1,ST1_Ignition_Status) ,XIC(Ignition_Bypass) ] ADD(OP220_Seq.CurrentStep,10,OP220_Seq.NextStep) OTU(Robot.CMD) ] ,XIO(OP220.DryCycle) XIC(AOI_CTS1.Program_Reject) [XIO(Ignition_Bypass) MOVE(-3,ST1_Ignition_Status) ,XIC(Ignition_Bypass) ] MOVE(7100,OP220_Seq.NextStep) ];
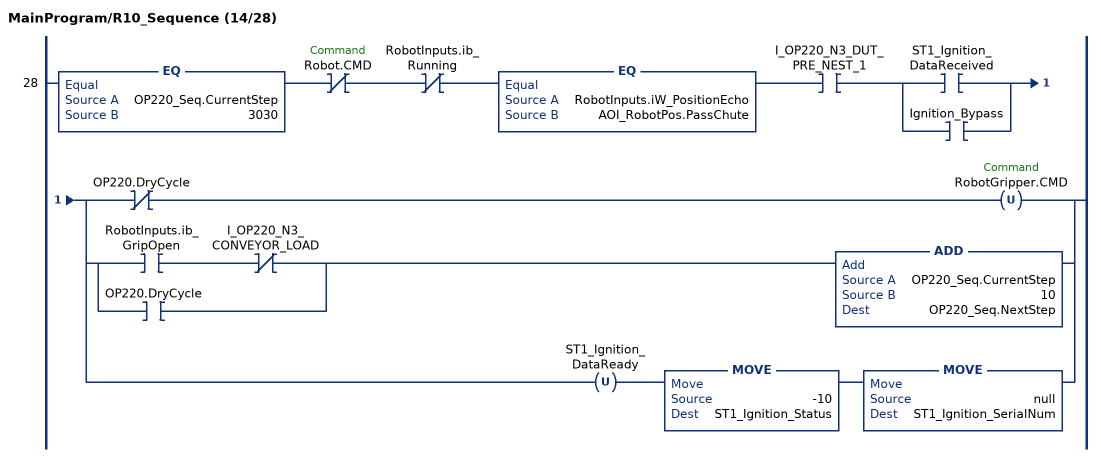
   28: EQ(OP220_Seq.CurrentStep,3030)XIO(Robot.CMD)XIO(RobotInputs.ib_Running)EQ(RobotInputs.iW_PositionEcho,AOI_RobotPos.PassChute)XIC(I_OP220_N3_DUT_PRE_NEST_1)[XIC(ST1_Ignition_DataReceived) ,XIC(Ignition_Bypass) ][XIO(OP220.DryCycle) OTU(RobotGripper.CMD) ,[XIC(RobotInputs.ib_GripOpen) XIO(I_OP220_N3_CONVEYOR_LOAD) ,XIC(OP220.DryCycle) ] ADD(OP220_Seq.CurrentStep,10,OP220_Seq.NextStep) ,OTU(ST1_Ignition_DataReady) MOVE(-10,ST1_Ignition_Status) MOVE(null,ST1_Ignition_SerialNum) ];
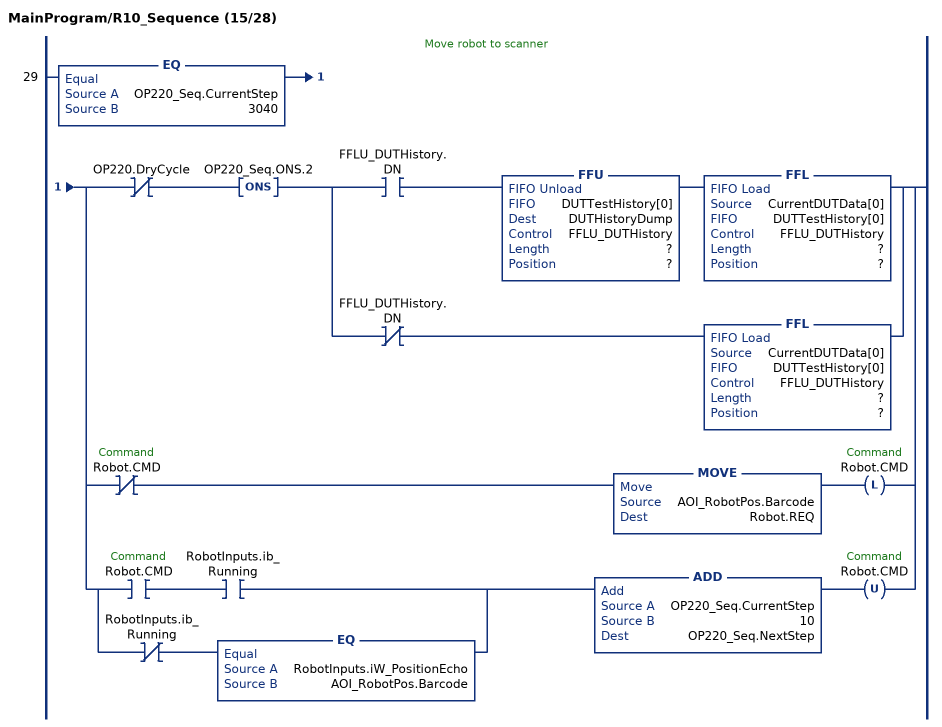
   // Move robot to scanner
   29: EQ(OP220_Seq.CurrentStep,3040)[XIO(OP220.DryCycle) ONS(OP220_Seq.ONS.2) [XIC(FFLU_DUTHistory.DN) FFU(DUTTestHistory[0],DUTHistoryDump,FFLU_DUTHistory,?,?) FFL(CurrentDUTData[0],DUTTestHistory[0],FFLU_DUTHistory,?,?) ,XIO(FFLU_DUTHistory.DN) FFL(CurrentDUTData[0],DUTTestHistory[0],FFLU_DUTHistory,?,?) ] ,XIO(Robot.CMD) MOVE(AOI_RobotPos.Barcode,Robot.REQ) OTL(Robot.CMD) ,[XIC(Robot.CMD) XIC(RobotInputs.ib_Running) ,XIO(RobotInputs.ib_Running) EQ(RobotInputs.iW_PositionEcho,AOI_RobotPos.Barcode) ] ADD(OP220_Seq.CurrentStep,10,OP220_Seq.NextStep) OTU(Robot.CMD) ];
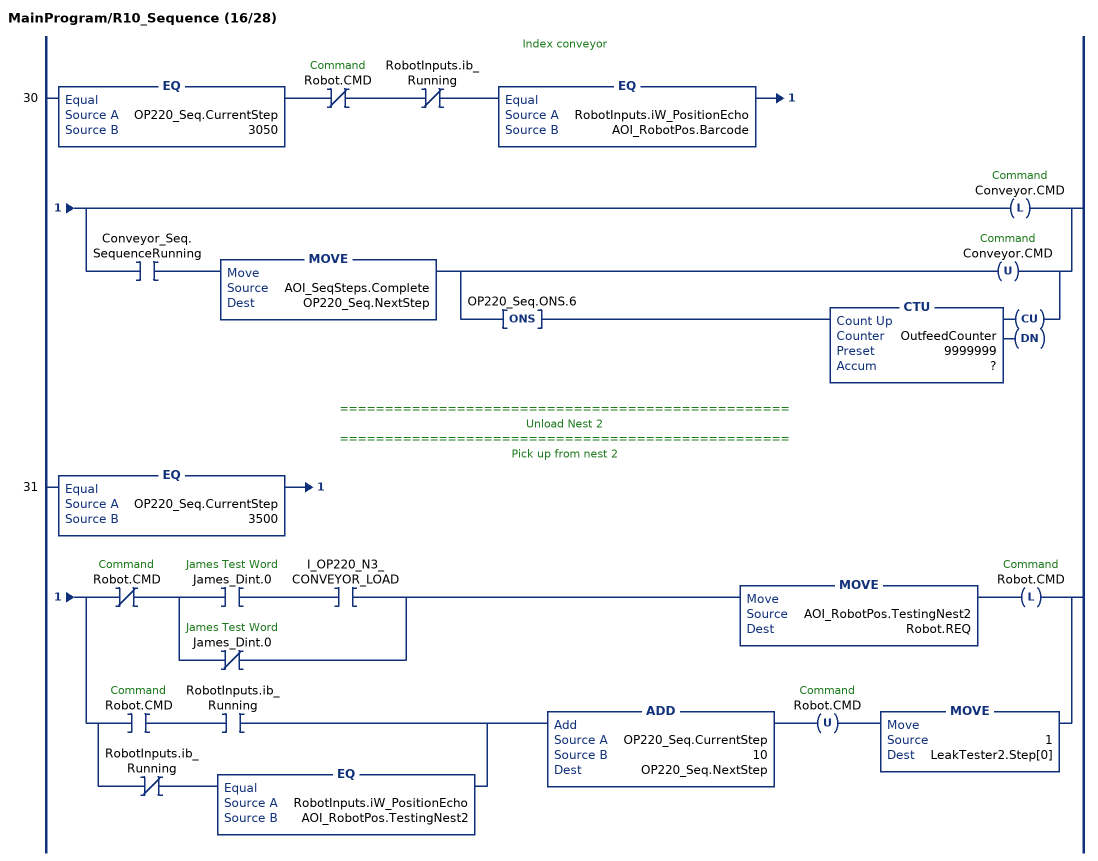
   // Index conveyor
   30: EQ(OP220_Seq.CurrentStep,3050)XIO(Robot.CMD)XIO(RobotInputs.ib_Running)EQ(RobotInputs.iW_PositionEcho,AOI_RobotPos.Barcode)[OTL(Conveyor.CMD) ,XIC(Conveyor_Seq.SequenceRunning) MOVE(AOI_SeqSteps.Complete,OP220_Seq.NextStep) [OTU(Conveyor.CMD) ,ONS(OP220_Seq.ONS.6) CTU(OutfeedCounter,?,?) ] ];
   // ==================================================
   // Unload Nest 2
   // ==================================================
   // Pick up from nest 2
   31: EQ(OP220_Seq.CurrentStep,3500)[XIO(Robot.CMD) [XIC(James_Dint.0) XIC(I_OP220_N3_CONVEYOR_LOAD) ,XIO(James_Dint.0) ] MOVE(AOI_RobotPos.TestingNest2,Robot.REQ) OTL(Robot.CMD) ,[XIC(Robot.CMD) XIC(RobotInputs.ib_Running) ,XIO(RobotInputs.ib_Running) EQ(RobotInputs.iW_PositionEcho,AOI_RobotPos.TestingNest2) ] ADD(OP220_Seq.CurrentStep,10,OP220_Seq.NextStep) OTU(Robot.CMD) MOVE(1,LeakTester2.Step[0]) ];
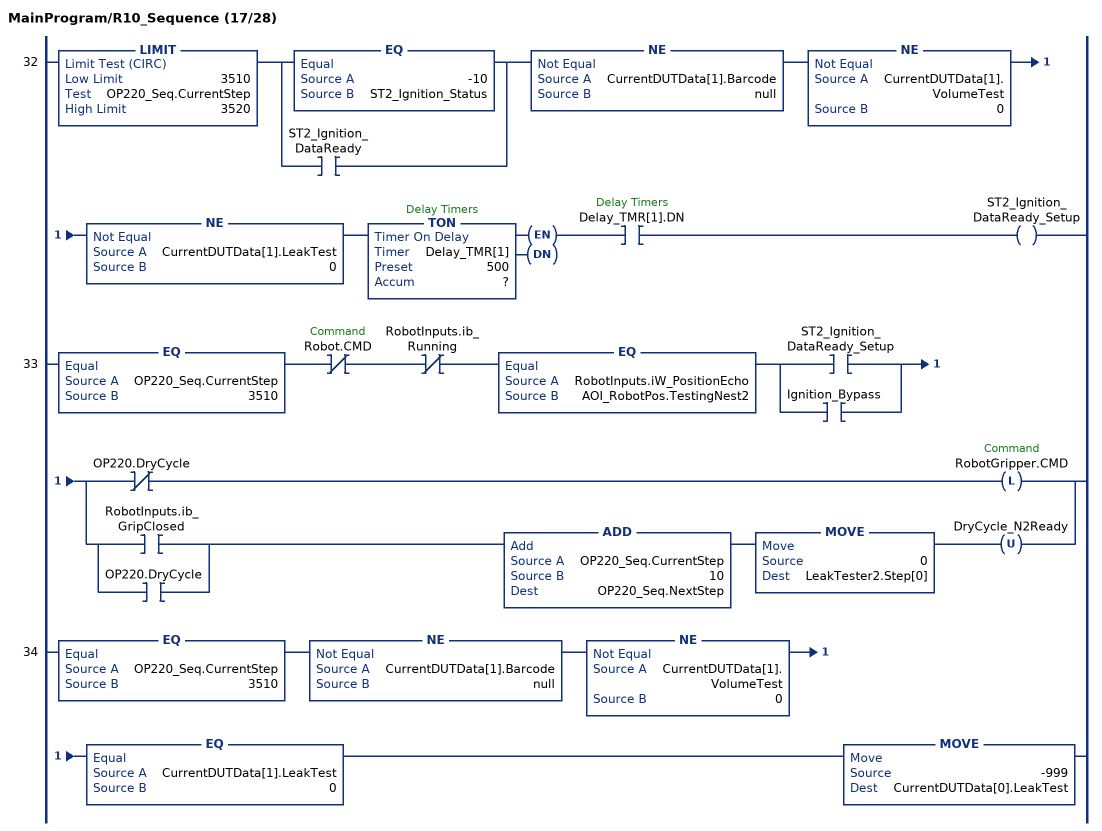
   32: LIMIT(3510,OP220_Seq.CurrentStep,3520)[EQ(-10,ST2_Ignition_Status) ,XIC(ST2_Ignition_DataReady) ]NE(CurrentDUTData[1].Barcode,null)NE(CurrentDUTData[1].VolumeTest,0)NE(CurrentDUTData[1].LeakTest,0)TON(Delay_TMR[1],?,?)XIC(Delay_TMR[1].DN)OTE(ST2_Ignition_DataReady_Setup);
   33: EQ(OP220_Seq.CurrentStep,3510)XIO(Robot.CMD)XIO(RobotInputs.ib_Running)EQ(RobotInputs.iW_PositionEcho,AOI_RobotPos.TestingNest2)[XIC(ST2_Ignition_DataReady_Setup) ,XIC(Ignition_Bypass) ][XIO(OP220.DryCycle) OTL(RobotGripper.CMD) ,[XIC(RobotInputs.ib_GripClosed) ,XIC(OP220.DryCycle) ] ADD(OP220_Seq.CurrentStep,10,OP220_Seq.NextStep) MOVE(0,LeakTester2.Step[0]) OTU(DryCycle_N2Ready) ];
   34: EQ(OP220_Seq.CurrentStep,3510)NE(CurrentDUTData[1].Barcode,null)NE(CurrentDUTData[1].VolumeTest,0)EQ(CurrentDUTData[1].LeakTest,0)MOVE(-999,CurrentDUTData[0].LeakTest);
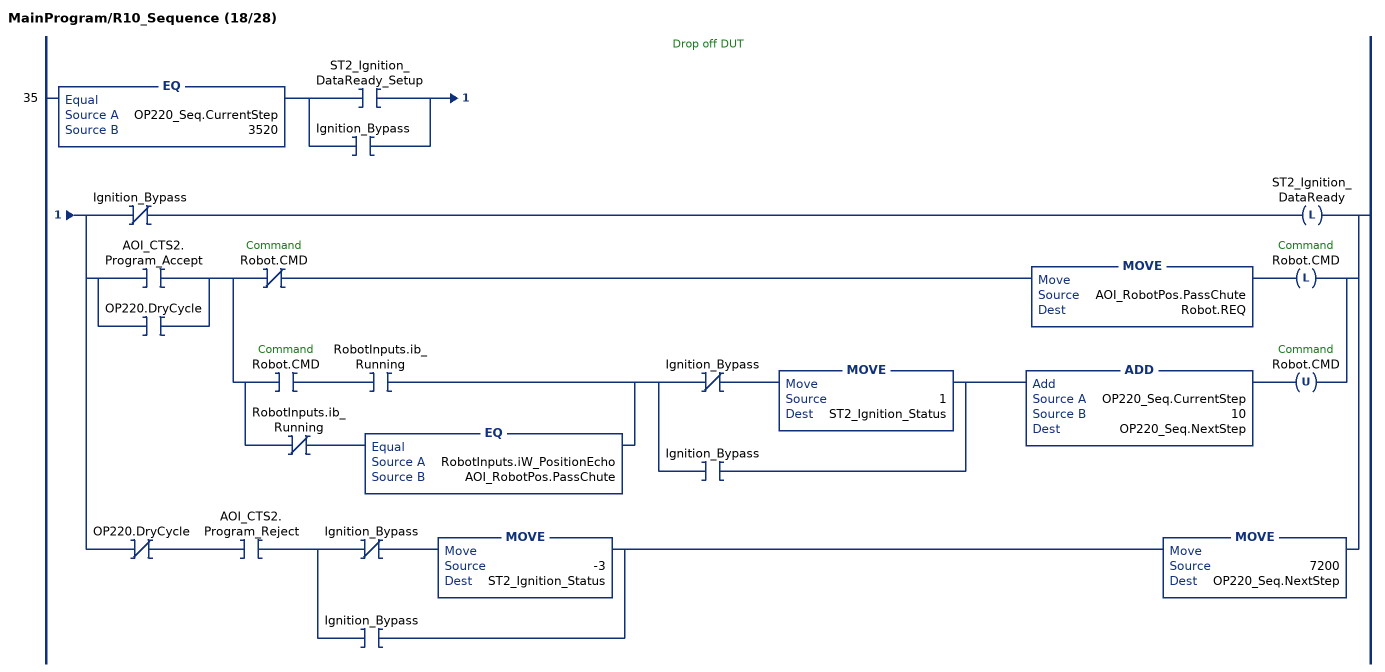
   // Drop off DUT
   35: EQ(OP220_Seq.CurrentStep,3520)[XIC(ST2_Ignition_DataReady_Setup) ,XIC(Ignition_Bypass) ][XIO(Ignition_Bypass) OTL(ST2_Ignition_DataReady) ,[XIC(AOI_CTS2.Program_Accept) ,XIC(OP220.DryCycle) ] [XIO(Robot.CMD) MOVE(AOI_RobotPos.PassChute,Robot.REQ) OTL(Robot.CMD) ,[XIC(Robot.CMD) XIC(RobotInputs.ib_Running) ,XIO(RobotInputs.ib_Running) EQ(RobotInputs.iW_PositionEcho,AOI_RobotPos.PassChute) ] [XIO(Ignition_Bypass) MOVE(1,ST2_Ignition_Status) ,XIC(Ignition_Bypass) ] ADD(OP220_Seq.CurrentStep,10,OP220_Seq.NextStep) OTU(Robot.CMD) ] ,XIO(OP220.DryCycle) XIC(AOI_CTS2.Program_Reject) [XIO(Ignition_Bypass) MOVE(-3,ST2_Ignition_Status) ,XIC(Ignition_Bypass) ] MOVE(7200,OP220_Seq.NextStep) ];
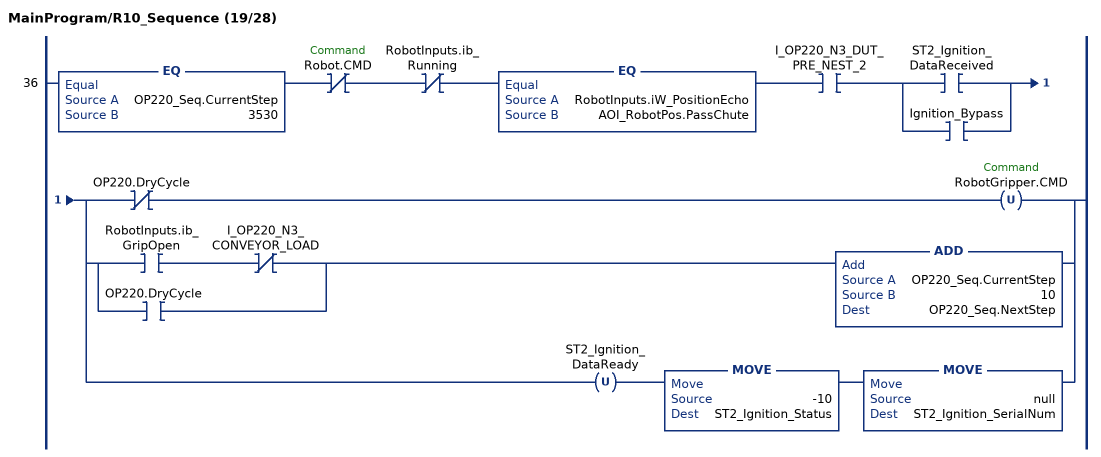
   36: EQ(OP220_Seq.CurrentStep,3530)XIO(Robot.CMD)XIO(RobotInputs.ib_Running)EQ(RobotInputs.iW_PositionEcho,AOI_RobotPos.PassChute)XIC(I_OP220_N3_DUT_PRE_NEST_2)[XIC(ST2_Ignition_DataReceived) ,XIC(Ignition_Bypass) ][XIO(OP220.DryCycle) OTU(RobotGripper.CMD) ,[XIC(RobotInputs.ib_GripOpen) XIO(I_OP220_N3_CONVEYOR_LOAD) ,XIC(OP220.DryCycle) ] ADD(OP220_Seq.CurrentStep,10,OP220_Seq.NextStep) ,OTU(ST2_Ignition_DataReady) MOVE(-10,ST2_Ignition_Status) MOVE(null,ST2_Ignition_SerialNum) ];
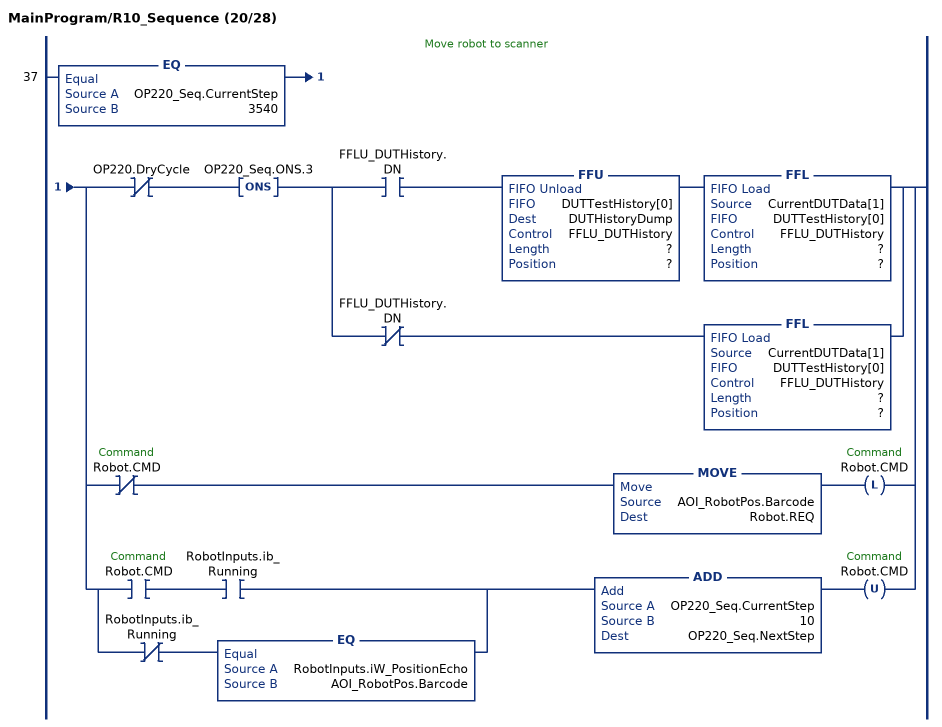
   // Move robot to scanner
   37: EQ(OP220_Seq.CurrentStep,3540)[XIO(OP220.DryCycle) ONS(OP220_Seq.ONS.3) [XIC(FFLU_DUTHistory.DN) FFU(DUTTestHistory[0],DUTHistoryDump,FFLU_DUTHistory,?,?) FFL(CurrentDUTData[1],DUTTestHistory[0],FFLU_DUTHistory,?,?) ,XIO(FFLU_DUTHistory.DN) FFL(CurrentDUTData[1],DUTTestHistory[0],FFLU_DUTHistory,?,?) ] ,XIO(Robot.CMD) MOVE(AOI_RobotPos.Barcode,Robot.REQ) OTL(Robot.CMD) ,[XIC(Robot.CMD) XIC(RobotInputs.ib_Running) ,XIO(RobotInputs.ib_Running) EQ(RobotInputs.iW_PositionEcho,AOI_RobotPos.Barcode) ] ADD(OP220_Seq.CurrentStep,10,OP220_Seq.NextStep) OTU(Robot.CMD) ];
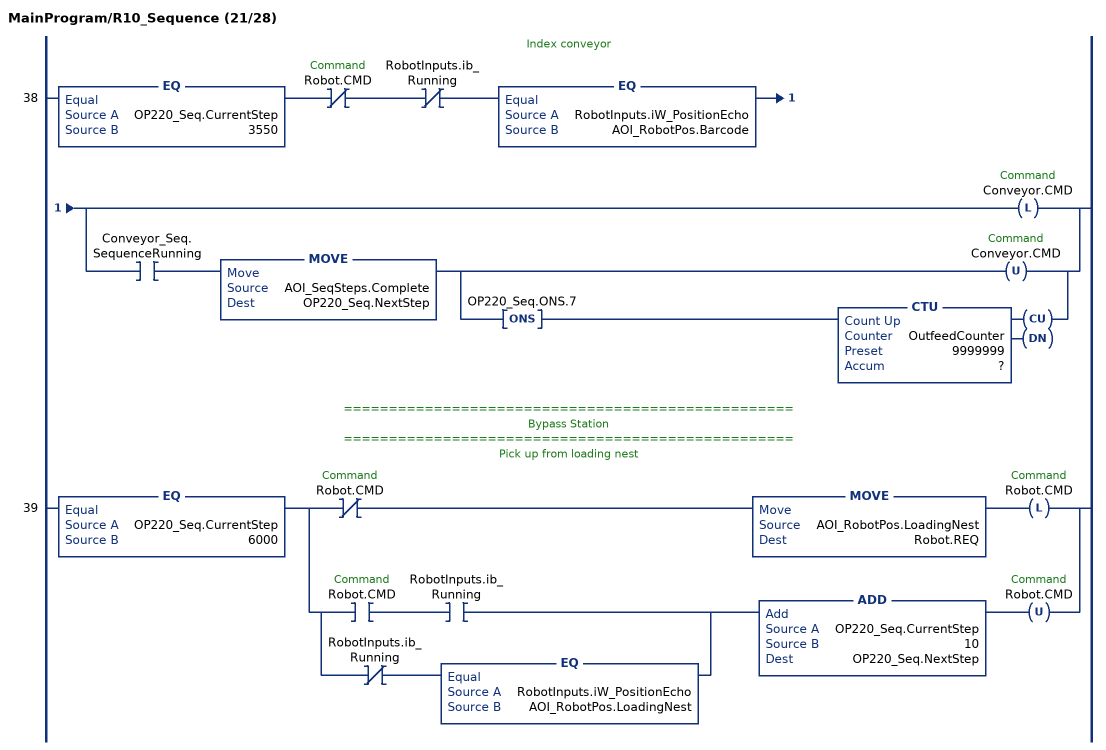
   // Index conveyor
   38: EQ(OP220_Seq.CurrentStep,3550)XIO(Robot.CMD)XIO(RobotInputs.ib_Running)EQ(RobotInputs.iW_PositionEcho,AOI_RobotPos.Barcode)[OTL(Conveyor.CMD) ,XIC(Conveyor_Seq.SequenceRunning) MOVE(AOI_SeqSteps.Complete,OP220_Seq.NextStep) [OTU(Conveyor.CMD) ,ONS(OP220_Seq.ONS.7) CTU(OutfeedCounter,?,?) ] ];
   // ==================================================
   // Bypass Station
   // ==================================================
   // Pick up from loading nest
   39: EQ(OP220_Seq.CurrentStep,6000)[XIO(Robot.CMD) MOVE(AOI_RobotPos.LoadingNest,Robot.REQ) OTL(Robot.CMD) ,[XIC(Robot.CMD) XIC(RobotInputs.ib_Running) ,XIO(RobotInputs.ib_Running) EQ(RobotInputs.iW_PositionEcho,AOI_RobotPos.LoadingNest) ] ADD(OP220_Seq.CurrentStep,10,OP220_Seq.NextStep) OTU(Robot.CMD) ];
